FUNCTION_BLOCK FB_ServoAxis ////Blok funkcyjny obslugujacy kompleksowao jedna Os 
VAR_INPUT	
	bSafetyReset			: BOOL;
	bEmergencyStop			: BOOL;	
	bInSafePosition			:BOOL;		
	I_TimeTableRef			: I_TimeTable255;
	sTTRowPreambule			: STRING;
	bELM_ChB				: BOOL;
END_VAR
VAR_OUTPUT
	nActEvent					: nAxis_ErrorList;
	udiActErrorCode				: UDINT;
END_VAR
VAR
	stInOuts					:st_Axis_InOuts;
	fbHomeSensorFTRIG			:F_TRIG;
	iCurrentPositionNumber		:USINT;
	bMoveAbsDone				:BOOL;
	bMoveModuloDone				:BOOL;
	bDirectHomingDone			:BOOL;
	bFullHomingDone				:BOOL;
	bQuickHomingRequest			:BOOL;

	bQuickHomingSynchLost		:BOOL;
	stHMI 						: ST_AxisHMI;
	i:USINT;
	lrPosition:LREAL;
	bCircularPositionsSet:BOOL;
	bMovementInterlock:BOOL;
	bPositionValid :BOOL;
	fbPositionValidTON:TON;
	tPositionValidDelay:TIME:=T#300MS;
	fbHomingSensorTON :TON;
	fbStepTON :TON;
	//OLD
	
	bEnableMotion				: BOOL;		// When TRUE - try to enable axis, when FALSE disable power - safeState
	bStandardSafetyDisable		: BOOL;     // Only safety reset required, No error
	McPower 					: MC_Power;
	McReset 					: MC_Reset;
	McStop	 					: MC_Stop;
	McHalt						: MC_Halt;
	McMoveAbs 					: MC_MoveAbsolute;
	McMoveModulo				: MC_MoveModulo;
	McMoveRel 					: MC_MoveRelative;
	McMoveVelocity	 			: MC_MoveVelocity;
	McJog	 					: MC_Jog;
	McReadActualPosition	 	: MC_ReadActualPosition;
	McReadActualVelocity	 	: MC_ReadActualVelocity;
	McHome						: MC_Home;
	McBrakeCtrl					: FB_BrakeControl;
	McTorqueMonitor				: FB_TorqueMonitoringEL_Ex2;
	McTorqueCtrl				: MC_TorqueControl;
	stHomimgParams				: ST_HomingOptions;
	bLimitSwitchMin: BOOL;
	bLimitSwitchMax: BOOL;
	iWorkStep_Axis: INT;
	fbTON_WorkStepTimeout: TON;
	bSetNewBrakeCtrl: BOOL;
	nAct_BrakeMode, nNew_BrakeMode: nHP_Axis_BrakeMode;
	fbFTRIG_BreakCtrlDone: F_TRIG;
	bTooglePowerState: BOOL;
	astErrorHistory: ARRAY [1..10] OF stErrorHistoryRow;
	fbEnableDelay	:TON;
	
END_VAR
VAR PERSISTENT
	lrReferencePositionAtHomeSensor: LREAL:=-1.0;
	lrLastPositionAtHomeSensor:LREAL:=-1.0;
	lrLastValidPositionValue:LREAL:=-1.0;
	stSettings				: ST_Axis_Settings;
END_VAR
VAR CONSTANT
	NUMBER_OF_PRESET_POSITIONS: USINT:=8;
END_VAR

stInOuts.bQ_SafetyRun :=TRUE;
stInOuts.bQ_SafetyErrorAck:=bSafetyReset;


// Read drive data
stInOuts.stAxis_Data.ReadStatus();
McReadActualPosition(Axis := stInOuts.stAxis_Data, Enable := TRUE);
McReadActualVelocity(Axis := stInOuts.stAxis_Data, Enable := TRUE);

iCurrentPositionNumber := 0;
IF prIsHomed AND prIsNotMoving THEN
	FOR i:=1 TO NUMBER_OF_PRESET_POSITIONS DO
		IF ABS(stSettings.arrPositions[i] - prCurrentPositionModulo) <= stSettings.lrPositionTolerance THEN
			iCurrentPositionNumber := i;
			EXIT;
		ELSIF stSettings.arrPositions[i] -stSettings.lrPositionTolerance <0 THEN
			IF 360.0 + (stSettings.arrPositions[i] -stSettings.lrPositionTolerance) <= prCurrentPositionModulo THEN
				iCurrentPositionNumber := i;
				EXIT;
			END_IF
		END_IF
	END_FOR
END_IF

//Servo position is valid
fbPositionValidTON(IN:= iCurrentPositionNumber <> 0 AND prIsInTargetPosition,PT:=tPositionValidDelay);
bPositionValid:= fbPositionValidTON.Q;
// Last Valid Position Value
IF prIsHomed AND prIsNotMoving AND prPositionValid THEN
	lrLastValidPositionValue := prCurrentPositionModulo;
ELSIF prIsMoving THEN 
	lrLastValidPositionValue := -1;
END_IF

//Read FB status
ACT_AxisFBs(); 	
ACT_AxisWorkSteps();


IF stSettings.bEN_CircularPositions AND NOT bCircularPositionsSet THEN
	lrPosition := 0.0;
	FOR i:=1 TO NUMBER_OF_PRESET_POSITIONS DO
		stSettings.arrPositions[i] := lrPosition;
		lrPosition := lrPosition + 360.0/NUMBER_OF_PRESET_POSITIONS;
	END_FOR
	bCircularPositionsSet:=TRUE;
END_IF


//Quick Homing
fbHomingSensorTON(IN:=stInOuts.bHomingSensor,PT:=T#300MS);
fbHomeSensorFTRIG(CLK:=fbHomingSensorTON.Q);
IF McMoveModulo.Busy AND prIsHomed AND fbHomeSensorFTRIG.Q AND stInOuts.stAxis_Data.Status.PositiveDirection THEN 
	mSavePositionAtHomeSensor();
	IF lrReferencePositionAtHomeSensor = -1.0 THEN
		lrReferencePositionAtHomeSensor := lrLastPositionAtHomeSensor;
	ELSE
		bQuickHomingRequest := stSettings.bEN_QuickHoming;
	END_IF
END_IF

//Manual Mode
IF stHMI.bDirectHomingRequest AND lrLastValidPositionValue >=0 THEN
	mDirectHoming(lrLastValidPositionValue);
ELSIF stHMI.bRequestStopAxis  THEN  
	mStopAxis();
ELSIF bQuickHomingRequest THEN
	mQuickHoming();
ELSIF prIsReady AND stHMI.bManualModeRequest THEN
	iWorkStep_Axis:=15;
END_IF

IF iWorkStep_Axis<>15 THEN
	stHMI.bJogBackwardButton := stHMI.bJogForwardButton := stHMI.bGoToSelectedPosition := FALSE;
END_IF


//HMI
stHMI.bIsReady := prIsReady;
stHMI.bIsHomed := prIsHomed;
stHMI.bIsMoving := prIsMoving;

stHMI.bRequestStopAxis := FALSE;
stHMI.bDirectHomingRequest :=FALSE;

ACTION ACT_AxisFBs:
bLimitSwitchMin	:= FALSE;
bLimitSwitchMax := FALSE;
// Power ON
IF stSettings.bEN_HW_LimitSwitches THEN
	IF NOT bELM_ChB THEN
		bLimitSwitchMin	:= NOT stInOuts.wI_DriveInfodata.0;
		bLimitSwitchMax	:= NOT stInOuts.wI_DriveInfodata.1;	
	ELSE
		bLimitSwitchMin	:= NOT stInOuts.wI_DriveInfodata.8;
		bLimitSwitchMax	:= NOT stInOuts.wI_DriveInfodata.9;	
	END_IF
END_IF
McPower(Axis:=stInOuts.stAxis_Data, Enable:=, Enable_Positive:=NOT bLimitSwitchMax, Enable_Negative:= (NOT bLimitSwitchMin OR McHome.Active));

// Error reset
McReset(Axis:=stInOuts.stAxis_Data);

// Homing
McHome(Axis := stInOuts.stAxis_Data, bCalibrationCam := stSettings.bEN_HomingSensor_Invert XOR stInOuts.bHomingSensor, Options := stHomimgParams);

// Stop FBs
McStop(Axis := stInOuts.stAxis_Data, Deceleration := 15000, Jerk := 100000);
McHalt(Axis := stInOuts.stAxis_Data, Deceleration := 15000, Jerk := 100000);
McBrakeCtrl(Axis := stInOuts.stAxis_Data);
fbFTRIG_BreakCtrlDone(CLK:= McBrakeCtrl.Busy);
IF fbFTRIG_BreakCtrlDone.Q THEN
	IF McBrakeCtrl.Mode = eBrakeMode_Automatic THEN	nAct_BrakeMode := nHP_Axis_BrakeMode.BrakeMode_Automatic;
	ELSIF McBrakeCtrl.Mode = eBrakeMode_Lock THEN nAct_BrakeMode := nHP_Axis_BrakeMode.BrakeMode_Lock;
	ELSIF McBrakeCtrl.Mode = eBrakeMode_Unlock THEN nAct_BrakeMode := nHP_Axis_BrakeMode.BrakeMode_Unlock;
	END_IF
END_IF
McBrakeCtrl.Execute := FALSE;
// Motion FBs

McJog(Axis := stInOuts.stAxis_Data, Mode := MC_JOGMODE_CONTINOUS, Acceleration := stSettings.rAcceleration, Deceleration := stSettings.rDeceleration, Jerk := 100000);
McMoveAbs(Axis := stInOuts.stAxis_Data, Acceleration := stSettings.rAcceleration, Deceleration := stSettings.rDeceleration, Jerk := 100000);
McMoveRel(Axis := stInOuts.stAxis_Data, Acceleration := stSettings.rAcceleration, Deceleration := stSettings.rDeceleration, Jerk := 100000);
McMoveVelocity(Axis := stInOuts.stAxis_Data, Acceleration := stSettings.rAcceleration, Deceleration := stSettings.rDeceleration, Jerk := 100000);
McMoveModulo(Axis := stInOuts.stAxis_Data, Acceleration := stSettings.rAcceleration, Deceleration := stSettings.rDeceleration, Jerk := 100000);
// Torque limitation
McTorqueMonitor( bCalculate:= bEnableMotion,
	rTorqueLimit:= ,
	Axis:= stInOuts.stAxis_Data);
McTorqueCtrl(Axis := stInOuts.stAxis_Data, Relative := FALSE, ContinuousUpdate := TRUE, TorqueRamp := 100);
END_ACTION

ACTION ACT_AxisWorkSteps:

IF NOT bEnableMotion AND iWorkStep_Axis < 90 THEN //Safety Stop
	IF bEmergencyStop AND prPositionValid AND bInSafePosition THEN
		iWorkStep_Axis:=90;
		bStandardSafetyDisable := TRUE;
	ELSE
		mNewEvent(nEvent := nAxis_ErrorList.STO_SignalActive, ErrorCode:= 0,bDisable:=TRUE);
	END_IF
	
ELSIF NOT prMovementExternalInterlock AND prIsMoving AND iWorkStep_Axis < 90 AND FALSE  THEN
	mNewEvent(nEvent := nAxis_ErrorList.MovementInterlockLost, ErrorCode:= 0,bDisable:=FALSE);
END_IF
bEnableMotion := stInOuts.bI_SS1_Release AND stInOuts.bI_STO_Release;

stSettings.rSlowSpeed_deg_s := LIMIT(1, stSettings.rSlowSpeed_deg_s, 50);
stSettings.rFastSpeed_deg_s := LIMIT(50, stSettings.rFastSpeed_deg_s, 300);
stSettings.rDeceleration := LIMIT(100, stSettings.rDeceleration, 5000);
stSettings.rAcceleration := LIMIT(100, stSettings.rAcceleration, 5000);

CASE iWorkStep_Axis OF
	0:	// Inicjalizacja
		mCancelAllCommands();
		bStandardSafetyDisable:=FALSE;
		iWorkStep_Axis := 1;
		
	1:	// Sprawdzenie parametrów pracy

		iWorkStep_Axis := 5;
		
	5: 	// Sprawdzenie gotowości do załączenia
		fbEnableDelay(PT:=T#3S,in:=bEnableMotion);
		McPower.Enable := fbEnableDelay.Q;
		IF McPower.Status THEN
			iWorkStep_Axis := 10;
		ELSIF McPower.Error THEN
			mNewEvent( nEvent := nAxis_ErrorList.MotionFB_Error,ErrorCode:= McPower.ErrorID,bDisable:=TRUE);
		END_IF
		
	10:	// Axis ready for new Cmds
		mCancelMoveCommands();
		IF prIsErrorActive THEN
			mNewEvent( nEvent := nAxis_ErrorList.MotionFB_Error,ErrorCode:= stInOuts.stAxis_Data.Status.ErrorID,bDisable:=TRUE);
		END_IF
		fbTON_WorkStepTimeout(IN:= FALSE);
		bMoveAbsDone := bDirectHomingDone:= bMoveModuloDone:= bFullHomingDone:= FALSE;
		
	15:	// Manual mode
		//Jog
		McJog.Velocity := stSettings.rSlowSpeed_deg_s/2;
		McJog(Axis := stInOuts.stAxis_Data, JogBackwards := stHMI.bJogBackwardButton, JogForward := stHMI.bJogForwardButton);
		//Positioning
		McMoveModulo.Direction:= MC_Direction.MC_Shortest_Way;
		McMoveModulo.Position := stSettings.arrPositions[LIMIT(1,stHMI.iManualPositionSelected,NUMBER_OF_PRESET_POSITIONS)];
		McMoveModulo.Velocity := stSettings.rSlowSpeed_deg_s;
		McMoveModulo.Execute:= stHMI.bGoToSelectedPosition;
		McHalt.Execute:=McMoveModulo.Active AND NOT stHMI.bGoToSelectedPosition;
		// Breake control
		IF bSetNewBrakeCtrl THEN
			McBrakeCtrl.Mode := nNew_BrakeMode;
			McBrakeCtrl.Execute := TRUE;	
			bSetNewBrakeCtrl := FALSE; 
		// Enable/disable axis
		ELSIF bTooglePowerState THEN
			McPower.Enable := NOT McPower.Enable;
 			bTooglePowerState := FALSE;
		ELSE
			McPower.Enable S= McJog.JogForward OR McJog.JogBackwards;
		END_IF	

		IF NOT stHMI.bManualModeRequest THEN
			iWorkStep_Axis:=10;
		END_IF
	
		
	20:	// Homing
		McHome.Execute := TRUE;
		IF McHome.Busy THEN
			iWorkStep_Axis := 21;	
		ELSIF McHome.Error THEN
			mNewEvent( nEvent := nAxis_ErrorList.MotionFB_Error,ErrorCode:= McHome.ErrorID,bDisable:=TRUE);
		END_IF
			
	21:	// Home done
		IF McHome.Done THEN
			bQuickHomingSynchLost := FALSE;
			McHome.Execute := FALSE;
			iWorkStep_Axis := 10;
			bFullHomingDone := TRUE;
//			//Move to first position
//			McMoveModulo.Direction:= MC_Direction.MC_Shortest_Way;
//			McMoveModulo.Position := stSettings.arrPositions[1];
//			McMoveModulo.Velocity := stSettings.rSlowSpeed_deg_s;
//			iWorkStep_Axis := 50;
			lrReferencePositionAtHomeSensor := -1;
		ELSIF McHome.Error THEN
			mNewEvent( nEvent := nAxis_ErrorList.MotionFB_Error,ErrorCode:= McHome.ErrorID,bDisable:=TRUE);
		ELSIF McHome.CommandAborted THEN
			mNewEvent(nEvent := nAxis_ErrorList.CommandAborted, ErrorCode:= McMoveModulo.ErrorID,bDisable:=TRUE);
		END_IF

		
	30:	// Move to absolute position
		McMoveAbs.Execute := TRUE;
		IF McMoveAbs.Busy THEN
			iWorkStep_Axis := 31;	
		ELSIF McMoveAbs.Error THEN
			mNewEvent(nEvent := nAxis_ErrorList.MotionFB_Error, ErrorCode:= McMoveAbs.ErrorID,bDisable:=TRUE);
		END_IF
	
	31:	// Move ABS done
		IF 	McMoveAbs.Done THEN
			McMoveAbs.Execute := FALSE;
			iWorkStep_Axis := 10;	
			bMoveAbsDone := TRUE;
		ELSIF McMoveAbs.Error THEN
			mNewEvent(nEvent := nAxis_ErrorList.MotionFB_Error, ErrorCode:= McMoveAbs.ErrorID,bDisable:=TRUE);
		ELSIF McMoveAbs.CommandAborted THEN	
			mNewEvent(nEvent := nAxis_ErrorList.CommandAborted, ErrorCode:= McMoveModulo.ErrorID,bDisable:=TRUE);
		END_IF
		
		
	40: //Direct Homing
		bQuickHomingRequest:=FALSE;
		McHome.HomingMode := MC_HomingMode.MC_Direct;
		McHome.Execute := TRUE;
		IF McHome.Busy THEN
			fbTON_WorkStepTimeout(IN:= FALSE);
			iWorkStep_Axis := 41;
		ELSIF McHome.Error THEN
			mNewEvent( nEvent := nAxis_ErrorList.MotionFB_Error,ErrorCode:= McHome.ErrorID,bDisable:=TRUE);
		END_IF
		
	41: //Direct Homing Done
		IF 	McHome.Done THEN
			iWorkStep_Axis := 10;	
			bDirectHomingDone := TRUE;
			McHome.Execute := FALSE;
		ELSIF McHome.Error THEN
			mNewEvent(nEvent := nAxis_ErrorList.MotionFB_Error, ErrorCode:= McHome.ErrorID,bDisable:=TRUE);
		ELSIF McHome.CommandAborted THEN
			mNewEvent(nEvent := nAxis_ErrorList.CommandAborted, ErrorCode:= McMoveModulo.ErrorID,bDisable:=TRUE);
		END_IF
	
	50:	// Move Modulo
		McMoveModulo.Execute := TRUE;
		IF McMoveModulo.Busy THEN
			iWorkStep_Axis := 51;		// Done
		ELSIF McMoveModulo.Error THEN
			mNewEvent(nEvent := nAxis_ErrorList.MotionFB_Error, ErrorCode:= McMoveModulo.ErrorID,bDisable:=TRUE);
		END_IF
	
	51:	// Move Modulo Done
		IF 	McMoveModulo.Done THEN
			iWorkStep_Axis := 10;	
			bMoveModuloDone := TRUE;
			McMoveModulo.Execute := FALSE;
		ELSIF McMoveModulo.Error THEN
			mNewEvent(nEvent := nAxis_ErrorList.MotionFB_Error, ErrorCode:= McMoveModulo.ErrorID,bDisable:=TRUE);
		ELSIF McMoveModulo.CommandAborted THEN
			mNewEvent(nEvent := nAxis_ErrorList.CommandAborted, ErrorCode:= McMoveModulo.ErrorID,bDisable:=TRUE);
		END_IF
		
	
	90:	// Error
		mCancelAllCommands();
		//fbStepTON(IN:=bStandardSafetyDisable, PT:=T#10S); 
		IF bStandardSafetyDisable AND stInOuts.bI_SS1_State AND stInOuts.bI_STO_State OR NOT bStandardSafetyDisable OR fbStepTON.Q  THEN
			iWorkStep_Axis := 91;
			fbStepTON(IN:=FALSE);
		END_IF
		

	91: // Stop 		
		McStop.Execute := TRUE;
		IF McStop.Done OR McStop.Error THEN
			McStop.Execute := FALSE;
			iWorkStep_Axis := 92;
		END_IF
		
	92: // Disable Power 
		McPower.Enable := FALSE;
		IF NOT McPower.Status THEN
			iWorkStep_Axis := 94;
		ELSIF McPower.Error THEN
			mNewEvent(nEvent := nAxis_ErrorList.MotionFB_Error, ErrorCode:= McPower.ErrorID,bDisable:=TRUE);
		END_IF
		
	93: // Stop No Disbale
		mCancelMoveCommands();
		McHalt.Execute := TRUE;
		IF McHalt.Done THEN
			iWorkStep_Axis:=94;
			McHalt.Execute := FALSE;
		ELSIF McHalt.Error THEN
			mNewEvent(nEvent := nAxis_ErrorList.MotionFB_Error, ErrorCode:= McHalt.ErrorID,bDisable:=TRUE);
		END_IF;
		
	94:	// Axis wait for reset
		McReset.Execute := FALSE;
		fbTON_WorkStepTimeout(IN:= FALSE);
		IF bStandardSafetyDisable AND bEnableMotion THEN
			iWorkStep_Axis := 96;
		END_IF
	
	95: // Axis reset
		IF stInOuts.stAxis_Data.Status.Error THEN
			iWorkStep_Axis := 96;
		ELSE
			iWorkStep_Axis := 97;
		END_IF
		
	96: // Perform Mc Reset
		McReset.Execute := TRUE;
		IF McReset.Done THEN	// Reset axis
			McReset.Execute := FALSE;
			fbTON_WorkStepTimeout(IN:= FALSE);
			iWorkStep_Axis := 97;
		ELSIF McReset.Error THEN	
			McReset.Execute := FALSE;
			mNewEvent(nEvent := nAxis_ErrorList.MotionFB_Error, ErrorCode:= McReset.ErrorID,bDisable:=TRUE);
		END_IF
		
	97:	// Reset succesfull
		nActEvent := nAxis_ErrorList.NoError;
		udiActErrorCode:= 0;
		fbTON_WorkStepTimeout(IN:= TRUE, PT:= T#40MS);
		IF fbTON_WorkStepTimeout.Q THEN
			fbTON_WorkStepTimeout(IN:= FALSE);
			iWorkStep_Axis := 0;
		END_IF
		
END_CASE
END_ACTION

METHOD mAddTimeStat : BOOL
VAR_INPUT
	sText 		: STRING(255);
END_VAR
VAR
	sTextTmp	: STRING(255);
END_VAR
IF I_TimeTableRef <> 0 THEN
	CONCAT2(pSrcString1 := ADR(sTTRowPreambule), pSrcString2 := ADR(sText), pDstString := ADR(sTextTmp), nDstSize := SIZEOF(sTextTmp));
	I_TimeTableRef.mPushText(sText := sTextTmp);
END_IF
END_METHOD

METHOD mCancelAllCommands : BOOL
VAR_INPUT
END_VAR
McPower.Enable := McReset.Execute := McHome.Execute := McStop.Execute := McHalt.Execute:=  FALSE;
mCancelMoveCommands();
END_METHOD

METHOD mCancelMoveCommands : BOOL
VAR_INPUT
END_VAR
McJog.JogForward := McJog.JogBackwards := McMoveAbs.Execute := McMoveRel.Execute := McMoveVelocity.Execute := McMoveModulo.Execute:=FALSE;
END_METHOD

METHOD mDirectHoming : BOOL
VAR_INPUT
	lrPositionToSet :LREAL;
END_VAR
VAR_OUTPUT
	bBusy		: BOOL;
	bError		: BOOL;
	udiErrorId	: UDINT;
END_VAR
mDirectHoming :=FALSE;
IF prIsReady THEN
	McHome.Position := lrPositionToSet;
	iWorkStep_Axis := 40;
ELSIF McHome.Error OR iWorkStep_Axis <40 OR iWorkStep_Axis >41  THEN
	mDirectHoming := TRUE;
	bError := TRUE;
	udiErrorId := INT_TO_UINT(iWorkStep_Axis);	
END_IF

bBusy := McHome.Busy;
IF bDirectHomingDone THEN
	mDirectHoming := TRUE;
	bDirectHomingDone :=FALSE;
END_IF;
udiErrorId := McHome.ErrorID;
END_METHOD

METHOD mErrorReset : BOOL
VAR_OUTPUT
	bError		: BOOL;
	udiErrorId	: UDINT;
END_VAR
IF iWorkStep_Axis = 94 THEN
	iWorkStep_Axis := 95;
END_IF
END_METHOD

METHOD mFullHoming : BOOL
VAR_INPUT
END_VAR
VAR_OUTPUT
	bBusy		: BOOL;
	bError		: BOOL;
	udiErrorId	: UDINT;
END_VAR
mFullHoming := FALSE;
IF prIsReady THEN
	iWorkStep_Axis := 20;
	McHome.Position := 357;
	McHome. HomingMode := MC_HomingMode.MC_DefaultHoming;
	stHomimgParams.SearchDirection := MC_Direction.MC_Positive_Direction;
	stHomimgParams.SyncDirection := MC_Direction.MC_Negative_Direction;
	stHomimgParams.SearchVelocity := 10.0;
	stHomimgParams.SyncVelocity := 1;
	stHomimgParams.ReferenceMode := E_EncoderReferenceMode.ENCODERREFERENCEMODE_DEFAULt;
ELSIF McHome.Error OR iWorkStep_Axis < 20 OR iWorkStep_Axis > 21 THEN
	mFullHoming := TRUE;
	bError := TRUE;
	udiErrorId := INT_TO_UINT(iWorkStep_Axis);	
END_IF

bBusy := McHome.Busy;
IF bFullHomingDone THEN
	mFullHoming := TRUE;
	bFullHomingDone :=FALSE;
END_IF;
udiErrorId := McHome.ErrorID;
END_METHOD

METHOD mMoveFastToPresetPos : BOOL
VAR_INPUT
	iPosNumber	:USINT;
	bFast:BOOL;
END_VAR
VAR_OUTPUT
	bBusy		: BOOL;
	bError		: BOOL;
	udiErrorId	: UDINT;
END_VAR
mMoveFastToPresetPos :=FALSE;
IF prIsReady AND prIsHomed THEN
	iPosNumber := MIN(20,iPosNumber);
	McMoveAbs.Position := stSettings.arrPositions[iPosNumber];
	IF bFast THEN
		McMoveAbs.Velocity := stSettings.rFastSpeed_deg_s;
	ELSE
		McMoveAbs.Velocity := stSettings.rSlowSpeed_deg_s;
	END_IF
	iWorkStep_Axis := 30;
ELSIF McMoveAbs.Error OR iWorkStep_Axis <30 OR iWorkStep_Axis >31  THEN
	mMoveFastToPresetPos := TRUE;
	bError := TRUE;
	udiErrorId := INT_TO_UINT(iWorkStep_Axis);	
END_IF

bBusy := McMoveAbs.Busy;
IF bMoveAbsDone THEN
	mMoveFastToPresetPos := TRUE;
	bMoveAbsDone :=FALSE;
END_IF;
END_METHOD

METHOD mMoveModuloToPosition : BOOL
VAR_INPUT
	iPosNumber	:USINT;
	bFast:BOOL;
END_VAR
VAR_OUTPUT
	bBusy		: BOOL;
	bError		: BOOL;
	bNotReady	: BOOL;
	udiErrorId	: UDINT;
END_VAR
mMoveModuloToPosition :=FALSE;
IF prIsReady AND prIsHomed THEN
	McMoveModulo.Direction:= MC_Direction.MC_Shortest_Way;
	iPosNumber := MIN(20,iPosNumber);
	McMoveModulo.Position := stSettings.arrPositions[iPosNumber];
	IF bFast THEN
		McMoveModulo.Velocity := stSettings.rFastSpeed_deg_s;
	ELSE
		McMoveModulo.Velocity := stSettings.rSlowSpeed_deg_s;
	END_IF
	iWorkStep_Axis := 50;	
ELSIF McMoveModulo.Error THEN
	mMoveModuloToPosition := TRUE;
	bError := TRUE;
	udiErrorId :=McMoveModulo.ErrorID;	
ELSIF iWorkStep_Axis <50 OR iWorkStep_Axis >51 THEN
	mMoveModuloToPosition := TRUE;
	bNotReady := TRUE;
	udiErrorId := INT_TO_UINT(iWorkStep_Axis);	
END_IF

bBusy := McMoveModulo.Busy;
IF bMoveModuloDone THEN
	mMoveModuloToPosition := TRUE;
	bMoveModuloDone :=FALSE;
END_IF;
END_METHOD

METHOD INTERNAL mNewEvent : BOOL
VAR_INPUT
	nEvent: nAxis_ErrorList;
	ErrorCode: UDINT;
	bDisable: BOOL;
END_VAR
bStandardSafetyDisable :=FALSE;
MEMMOVE(srcAddr:= ADR(astErrorHistory[1]), destAddr := ADR(astErrorHistory[2]), n:= 9* SIZEOF(astErrorHistory[1]));
astErrorHistory[1].tTimeStamp := TIME();
astErrorHistory[1].sDescription := TO_STRING(nEvent);
astErrorHistory[1].iWorkStep1 := iWorkStep_Axis;
astErrorHistory[1].udiErrorCode := ErrorCode;
IF bDisable THEN
	iWorkStep_Axis := 90;
ELSE
	iWorkStep_Axis := 93;
END_IF
nActEvent := nEvent;
udiActErrorCode:= ErrorCode;
END_METHOD

METHOD mQuickHoming : BOOL

VAR_OUTPUT
	bBusy		: BOOL;
	bError		: BOOL;
	udiErrorId	: UDINT;
END_VAR
mQuickHoming :=FALSE;
IF prIsReady AND prIsHomed AND lrReferencePositionAtHomeSensor >= 0 AND lrLastPositionAtHomeSensor >= 0 THEN
	IF ABS(lrReferencePositionAtHomeSensor - lrLastPositionAtHomeSensor) > 1.0 THEN
		mNewEvent( nEvent := nAxis_ErrorList.QuickHomingError,ErrorCode:= McHome.ErrorID,bDisable:=FALSE);
		bQuickHomingSynchLost :=TRUE;
		bQuickHomingRequest:=FALSE;
	ELSE
		mDirectHoming(prCurrentPositionModulo + (lrReferencePositionAtHomeSensor - lrLastPositionAtHomeSensor));
	END_IF
END_IF
END_METHOD

METHOD mSavePositionAtHomeSensor : BOOL
VAR_INPUT
END_VAR
IF prCurrentPositionModulo <> -1 THEN
	lrLastPositionAtHomeSensor:=prCurrentPositionModulo;
END_IF;
END_METHOD

METHOD mStopAxis : BOOL
VAR_INPUT
END_VAR
mNewEvent(nEvent := nAxis_ErrorList.CommandAborted, ErrorCode:= 0,bDisable:=FALSE);
mStopAxis:=TRUE;
END_METHOD

{attribute 'monitoring' := 'call'}
PROPERTY prActualPosition : LREAL
GET
IF McReadActualPosition.Valid AND prIsHomed THEN		
	prActualPosition := McReadActualPosition.Position;
ELSE
	prActualPosition := -1;
END_IF
END_GET
END_PROPERTY

{attribute 'monitoring' := 'call'}
PROPERTY prActualVelocity : LREAL
GET
IF McReadActualVelocity.Valid THEN
	prActualVelocity := McReadActualVelocity.ActualVelocity;
ELSE
	prActualVelocity := -1;
END_IF
END_GET
END_PROPERTY

{attribute 'monitoring' := 'call'}
PROPERTY prCurrentPositionModulo : LREAL
GET
IF McReadActualPosition.Valid AND prIsHomed THEN		
	prCurrentPositionModulo := stInOuts.stAxis_Data.NcToPlc.ModuloActPos;
ELSE
	prCurrentPositionModulo := -1;
END_IF
END_GET
END_PROPERTY

{attribute 'monitoring' := 'call'}
PROPERTY prCurrentPositionNumber : USINT
GET
prCurrentPositionNumber:=iCurrentPositionNumber;
END_GET
END_PROPERTY

{attribute 'monitoring' := 'call'}
PROPERTY prEnabled : BOOL
GET
prEnabled:= McPower.Status;
END_GET
END_PROPERTY

{attribute 'monitoring' := 'call'}
PROPERTY prIsErrorActive : BOOL
GET
prIsErrorActive := stInOuts.stAxis_Data.Status.Error OR (iWorkStep_Axis >= 90 AND NOT bStandardSafetyDisable);
END_GET
END_PROPERTY

{attribute 'monitoring' := 'call'}
PROPERTY prIsHomed : BOOL
GET
prIsHomed := stInOuts.stAxis_Data.Status.Homed AND NOT bQuickHomingSynchLost;
END_GET
END_PROPERTY

{attribute 'monitoring' := 'call'}
PROPERTY prIsInTargetPosition : BOOL
GET
prIsInTargetPosition := stInOuts.stAxis_Data.Status.InTargetPosition;
END_GET
END_PROPERTY

{attribute 'monitoring' := 'call'}
PROPERTY prIsMoving : BOOL
GET
prIsMoving := stInOuts.stAxis_Data.Status.Moving;
END_GET
END_PROPERTY

{attribute 'monitoring' := 'call'}
PROPERTY prIsNotMoving : BOOL
GET
prIsNotMoving :=  stInOuts.stAxis_Data.Status.NotMoving;
END_GET
END_PROPERTY

{attribute 'monitoring' := 'call'}
PROPERTY prIsReady : BOOL
GET
prIsReady := stInOuts.stAxis_Data.Status.Operational AND NOT stInOuts.stAxis_Data.Status.Error AND McPower.Status AND iWorkStep_Axis = 10 AND prMovementExternalInterlock;
END_GET
END_PROPERTY

{attribute 'monitoring' := 'call'}
PROPERTY prMovementExternalInterlock : BOOL
GET
prMovementExternalInterlock:=bMovementInterlock;
END_GET
SET
bMovementInterlock:=prMovementExternalInterlock;
END_SET
END_PROPERTY

{attribute 'monitoring' := 'call'}
PROPERTY prPositionValid : BOOL
GET
prPositionValid:=bPositionValid;
END_GET
END_PROPERTY

END_FUNCTION_BLOCK

(* stored: Version 1.1.0.1, ProductVersion 3.1.4024.15
   POU FB_ServoAxis: Id {3057f7b8-ac98-4f2d-b555-83dd6c315250}, SpecialFunc None
   Folder Methods: Id {86110dc1-c583-424f-8e1a-53f0e16b101e}
   Folder Properties: Id {8dc25682-5df1-487c-935d-d480b60343c3}
   Action ACT_AxisFBs: Id {1733d200-0c8f-4641-80db-f206791f3515}
   Action ACT_AxisWorkSteps: Id {24332e8c-4fda-4b2a-bd2c-6d7b94bd461c}
   Method mAddTimeStat: Id {ab5ac6de-4b6f-4492-81c5-0cd32a15380e}
   Method mCancelAllCommands: Id {db48a037-4fb7-41cd-b68f-6707abdc91b7}
   Method mCancelMoveCommands: Id {acbb3440-cf87-41ac-a152-8968e26cb810}
   Method mDirectHoming: Id {d16f9285-8ee7-48c8-834a-f39aff3bc7b6}
   Method mErrorReset: Id {4c71a6d0-2eb8-4fd5-9ef2-16b78ed57f34}
   Method mFullHoming: Id {a262032b-63e5-4e87-a4b0-e16a24b03a3b}
   Method mMoveFastToPresetPos: Id {17b7a812-32ab-4488-9109-06aa0299f113}
   Method mMoveModuloToPosition: Id {b9786ee7-83c2-4602-a755-a5d8da1d53c5}
   Method mNewEvent: Id {45dc65cc-cc78-49f4-a976-6b04a137582d}
   Method mQuickHoming: Id {5b03c9ef-9972-4bbe-81ff-bccad90f604c}
   Method mSavePositionAtHomeSensor: Id {3a59daed-c1be-449e-8865-4c1bfb4a7379}
   Method mStopAxis: Id {09d463fc-b21d-48e3-8ec5-8c22313c676f}
   Property prActualPosition: Id {f40194ba-8306-4aaa-b5b5-5fb0758d9b45}
   Get Get: Id {8bac339c-d060-4766-ad8b-fd8c908a3488}
   Property prActualVelocity: Id {ff223880-cd07-4f47-8533-6780d3523a7c}
   Get Get: Id {78818ba6-1efe-447e-8266-54cd48988813}
   Property prCurrentPositionModulo: Id {a7f3473b-83b3-4341-bc35-77febc0fdef3}
   Get Get: Id {79826043-5518-4c9c-8b03-0cb607eb68d1}
   Property prCurrentPositionNumber: Id {ea3d6f95-12cc-4ac1-9e24-d1e623d6380c}
   Get Get: Id {5c223598-c8c8-44d8-8e1f-7aaddfe49b9a}
   Property prEnabled: Id {20ee9f61-720c-40a2-84c5-331a0b62253a}
   Get Get: Id {6f777018-1d15-4443-86fe-bcc9014295bc}
   Property prIsErrorActive: Id {da3f3089-581e-41ca-8bcd-c78e51817caa}
   Get Get: Id {436b39d5-59d0-48e6-8f59-40a1bc78273a}
   Property prIsHomed: Id {f71d9df2-615f-49d5-9f8f-a7959eb3e890}
   Get Get: Id {214f06e1-9c57-412c-bce6-1826f7c03c7d}
   Property prIsInTargetPosition: Id {7c58df86-0d69-4a2c-830b-ded4fd793ede}
   Get Get: Id {e786766e-c47f-4a16-8b97-2ac914454196}
   Property prIsMoving: Id {d921ac5b-ba42-4853-9806-c4dcb58d889c}
   Get Get: Id {f68ebf89-02ea-47cb-8cf6-53ef2c6e6de6}
   Property prIsNotMoving: Id {55c0575a-37a0-40ed-985f-602114fa2c8e}
   Get Get: Id {cb1572cd-ba6b-409d-8282-8e38c003a699}
   Property prIsReady: Id {6e65633e-98e6-41e4-9524-0f21768d5334}
   Get Get: Id {4e0e5a66-9481-4905-b577-efae5ddc6ef5}
   Property prMovementExternalInterlock: Id {3b41f782-19d6-4140-8d2f-1b560d59e4d3}
   Get Get: Id {48dd8a24-9dee-4b4f-bea6-609d20afc7b2}
   Set Set: Id {ba5d0f7e-ab05-44f9-94f9-be69fe117f78}
   Property prPositionValid: Id {8bd3caab-2706-4652-9796-d1cef13b5dc9}
   Get Get: Id {de089de8-ae53-46f8-95a8-55578f05c046} *)
